// TIA Portal V19 export
TYPE "LEXCHANGETRAY_typeEmActionPlastic"
// stored: Access Published
   STRUCT
      em6 : Bool;
      em5 : Bool;
   END_STRUCT;
END_TYPE
